// TIA Portal V19 export
FUNCTION "CollectAlarms" : Void   // FC62, LAD
TITLE = Alarm Collector Unit
// Collects alarms from the respective level and categorises the alarms into the different alarm classes. Filling the alarm DB with specific alarm messages which are defined in the comment of the defined alarm. The definition of possible alarms within a equipment is handled here.
// stored: Namespace Unit3.EM1, SetENOAutomatically false
   VAR_INPUT
      resetAlarms : Bool;
      disableAlarms : Bool;
   END_VAR
   VAR_OUTPUT
      commandsToUnit : "LUC_typeStateCommands";   // Feedback to the unit
   END_VAR
   VAR_TEMP   // added for the SCL form of the ladder/FBD networks
      _w1 : Bool;
   END_VAR
BEGIN

REGION Network 1: Reset Alarms
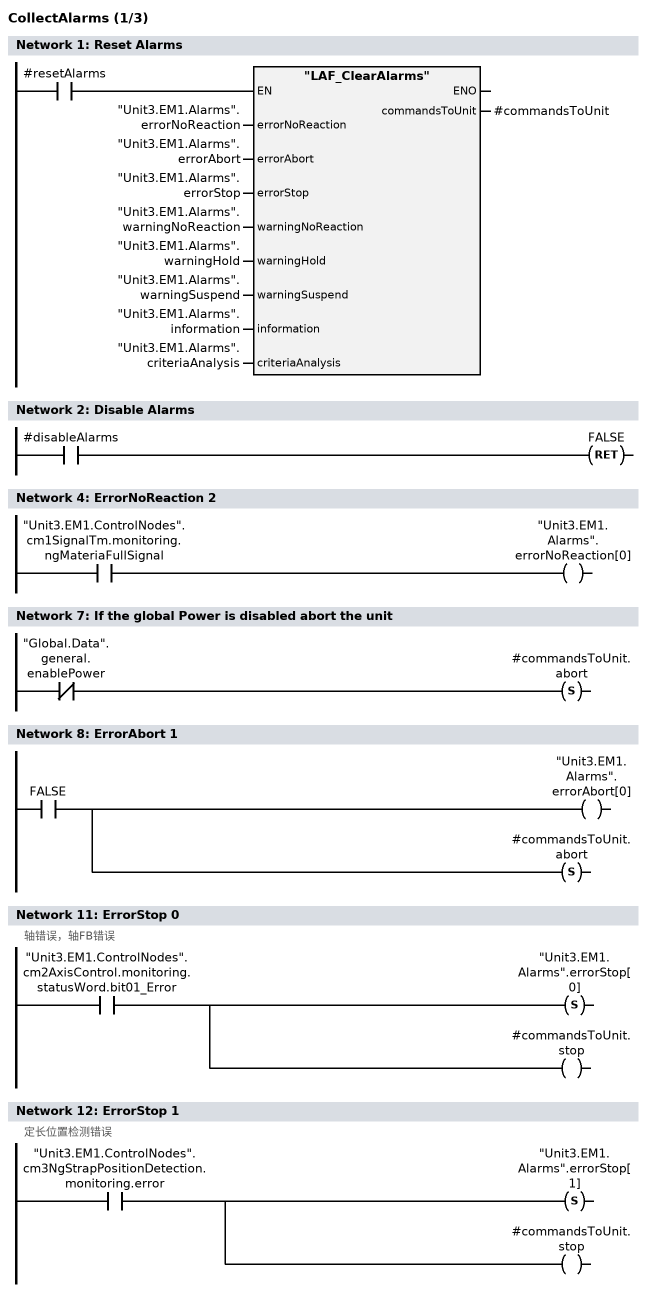
   RUNG wire#powerrail
      Contact( #resetAlarms )
      "LAF_ClearAlarms"(errorNoReaction := "Unit3.EM1.Alarms".errorNoReaction, errorAbort := "Unit3.EM1.Alarms".errorAbort, errorStop := "Unit3.EM1.Alarms".errorStop, warningNoReaction := "Unit3.EM1.Alarms".warningNoReaction, warningHold := "Unit3.EM1.Alarms".warningHold, warningSuspend := "Unit3.EM1.Alarms".warningSuspend, information := "Unit3.EM1.Alarms".information, criteriaAnalysis := "Unit3.EM1.Alarms".criteriaAnalysis, commandsToUnit => #commandsToUnit)
   END_RUNG
   // the same network as SCL:
   IF #resetAlarms THEN
       "LAF_ClearAlarms"(errorNoReaction := "Unit3.EM1.Alarms".errorNoReaction,
                         errorAbort := "Unit3.EM1.Alarms".errorAbort,
                         errorStop := "Unit3.EM1.Alarms".errorStop,
                         warningNoReaction := "Unit3.EM1.Alarms".warningNoReaction,
                         warningHold := "Unit3.EM1.Alarms".warningHold,
                         warningSuspend := "Unit3.EM1.Alarms".warningSuspend,
                         information := "Unit3.EM1.Alarms".information,
                         criteriaAnalysis := "Unit3.EM1.Alarms".criteriaAnalysis,
                         commandsToUnit => #commandsToUnit);
   END_IF;
END_REGION

REGION Network 2: Disable Alarms
   RUNG wire#powerrail
      Contact( #disableAlarms )
      ReturnCoil( FALSE )
   END_RUNG
   // the same network as SCL:
   IF #disableAlarms THEN
       ENO := FALSE;
       RETURN;
   END_IF;
END_REGION

REGION Network 3: *************** Error No Reaction ************************
END_REGION

REGION Network 4: ErrorNoReaction 2
   RUNG wire#powerrail
      Contact( "Unit3.EM1.ControlNodes".cm1SignalTm.monitoring.ngMateriaFullSignal )
      Coil( "Unit3.EM1.Alarms".errorNoReaction[0] )
   END_RUNG
   // the same network as SCL:
   "Unit3.EM1.Alarms".errorNoReaction[0] := "Unit3.EM1.ControlNodes".cm1SignalTm.monitoring.ngMateriaFullSignal;
END_REGION

REGION Network 6: *************** Error and Abort **************************
END_REGION

REGION Network 7: If the global Power is disabled abort the unit
   RUNG wire#powerrail
      I_Contact( "Global.Data".general.enablePower )
      S_Coil( #commandsToUnit.abort )
   END_RUNG
   // the same network as SCL:
   IF NOT "Global.Data".general.enablePower THEN #commandsToUnit.abort := TRUE; END_IF;
END_REGION

REGION Network 8: ErrorAbort 1
   RUNG wire#powerrail
      Contact( FALSE )
      wire#w1
      Coil( "Unit3.EM1.Alarms".errorAbort[0] )
   END_RUNG
   RUNG wire#w1
      S_Coil( #commandsToUnit.abort )
   END_RUNG
   // the same network as SCL:
   "Unit3.EM1.Alarms".errorAbort[0] := FALSE;
   IF FALSE THEN #commandsToUnit.abort := TRUE; END_IF;
END_REGION

REGION Network 10: *************** Error and Stop ***************************
END_REGION

REGION Network 11: ErrorStop 0
   // 轴错误，轴FB错误
   RUNG wire#powerrail
      Contact( "Unit3.EM1.ControlNodes".cm2AxisControl.monitoring.statusWord.bit01_Error )
      wire#w1
      S_Coil( "Unit3.EM1.Alarms".errorStop[0] )
   END_RUNG
   RUNG wire#w1
      Coil( #commandsToUnit.stop )
   END_RUNG
   // the same network as SCL:
   IF "Unit3.EM1.ControlNodes".cm2AxisControl.monitoring.statusWord.bit01_Error THEN
       "Unit3.EM1.Alarms".errorStop[0] := TRUE;
   END_IF;
   #commandsToUnit.stop := "Unit3.EM1.ControlNodes".cm2AxisControl.monitoring.statusWord.bit01_Error;
END_REGION

REGION Network 12: ErrorStop 1
   // 定长位置检测错误
   RUNG wire#powerrail
      Contact( "Unit3.EM1.ControlNodes".cm3NgStrapPositionDetection.monitoring.error )
      wire#w1
      S_Coil( "Unit3.EM1.Alarms".errorStop[1] )
   END_RUNG
   RUNG wire#w1
      Coil( #commandsToUnit.stop )
   END_RUNG
   // the same network as SCL:
   IF "Unit3.EM1.ControlNodes".cm3NgStrapPositionDetection.monitoring.error THEN
       "Unit3.EM1.Alarms".errorStop[1] := TRUE;
   END_IF;
   #commandsToUnit.stop := "Unit3.EM1.ControlNodes".cm3NgStrapPositionDetection.monitoring.error;
END_REGION

REGION Network 13: ErrorStop 2
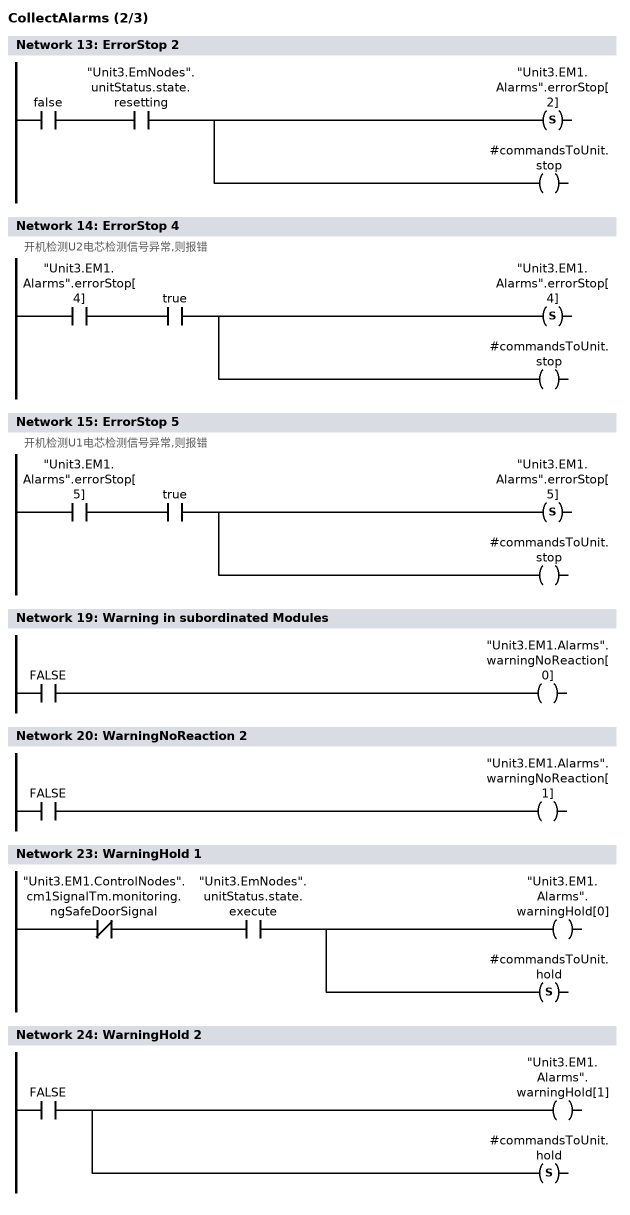
   RUNG wire#powerrail
      Contact( false )
      Contact( "Unit3.EmNodes".unitStatus.state.resetting )
      wire#w1
      S_Coil( "Unit3.EM1.Alarms".errorStop[2] )
   END_RUNG
   RUNG wire#w1
      Coil( #commandsToUnit.stop )
   END_RUNG
   // the same network as SCL:
   #_w1 := false AND "Unit3.EmNodes".unitStatus.state.resetting;
   IF #_w1 THEN "Unit3.EM1.Alarms".errorStop[2] := TRUE; END_IF;
   #commandsToUnit.stop := #_w1;
END_REGION

REGION Network 14: ErrorStop 4
   // 开机检测U2电芯检测信号异常,则报错
   RUNG wire#powerrail
      Contact( "Unit3.EM1.Alarms".errorStop[4] )
      Contact( true )
      wire#w1
      S_Coil( "Unit3.EM1.Alarms".errorStop[4] )
   END_RUNG
   RUNG wire#w1
      Coil( #commandsToUnit.stop )
   END_RUNG
   // the same network as SCL:
   #_w1 := "Unit3.EM1.Alarms".errorStop[4] AND true;
   IF #_w1 THEN "Unit3.EM1.Alarms".errorStop[4] := TRUE; END_IF;
   #commandsToUnit.stop := #_w1;
END_REGION

REGION Network 15: ErrorStop 5
   // 开机检测U1电芯检测信号异常,则报错
   RUNG wire#powerrail
      Contact( "Unit3.EM1.Alarms".errorStop[5] )
      Contact( true )
      wire#w1
      S_Coil( "Unit3.EM1.Alarms".errorStop[5] )
   END_RUNG
   RUNG wire#w1
      Coil( #commandsToUnit.stop )
   END_RUNG
   // the same network as SCL:
   #_w1 := "Unit3.EM1.Alarms".errorStop[5] AND true;
   IF #_w1 THEN "Unit3.EM1.Alarms".errorStop[5] := TRUE; END_IF;
   #commandsToUnit.stop := #_w1;
END_REGION

REGION Network 18: *************** Warning No Reaction **********************
END_REGION

REGION Network 19: Warning in subordinated Modules
   RUNG wire#powerrail
      Contact( FALSE )
      Coil( "Unit3.EM1.Alarms".warningNoReaction[0] )
   END_RUNG
   // the same network as SCL:
   "Unit3.EM1.Alarms".warningNoReaction[0] := FALSE;
END_REGION

REGION Network 20: WarningNoReaction 2
   RUNG wire#powerrail
      Contact( FALSE )
      Coil( "Unit3.EM1.Alarms".warningNoReaction[1] )
   END_RUNG
   // the same network as SCL:
   "Unit3.EM1.Alarms".warningNoReaction[1] := FALSE;
END_REGION

REGION Network 22: *************** Warning Hold **************************
END_REGION

REGION Network 23: WarningHold 1
   RUNG wire#powerrail
      I_Contact( "Unit3.EM1.ControlNodes".cm1SignalTm.monitoring.ngSafeDoorSignal )
      Contact( "Unit3.EmNodes".unitStatus.state.execute )
      wire#w1
      Coil( "Unit3.EM1.Alarms".warningHold[0] )
   END_RUNG
   RUNG wire#w1
      S_Coil( #commandsToUnit.hold )
   END_RUNG
   // the same network as SCL:
   "Unit3.EM1.Alarms".warningHold[0] := NOT "Unit3.EM1.ControlNodes".cm1SignalTm.monitoring.ngSafeDoorSignal AND "Unit3.EmNodes".unitStatus.state.execute;
   IF NOT "Unit3.EM1.ControlNodes".cm1SignalTm.monitoring.ngSafeDoorSignal AND "Unit3.EmNodes".unitStatus.state.execute THEN
       #commandsToUnit.hold := TRUE;
   END_IF;
END_REGION

REGION Network 24: WarningHold 2
   RUNG wire#powerrail
      Contact( FALSE )
      wire#w1
      Coil( "Unit3.EM1.Alarms".warningHold[1] )
   END_RUNG
   RUNG wire#w1
      S_Coil( #commandsToUnit.hold )
   END_RUNG
   // the same network as SCL:
   "Unit3.EM1.Alarms".warningHold[1] := FALSE;
   IF FALSE THEN #commandsToUnit.hold := TRUE; END_IF;
END_REGION

REGION Network 26: *************** Warning Suspend ***********************
END_REGION

REGION Network 27: WarningSuspend 1
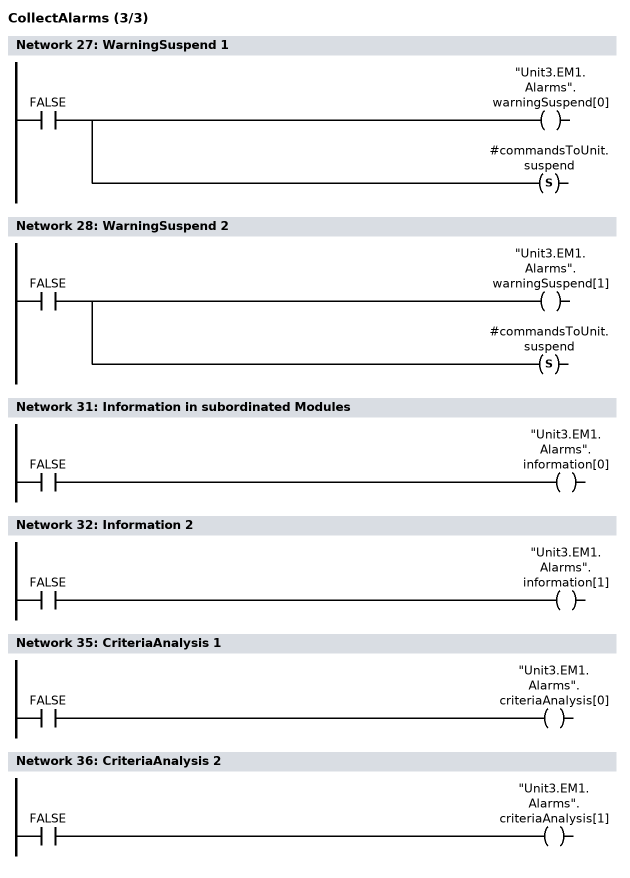
   RUNG wire#powerrail
      Contact( FALSE )
      wire#w1
      Coil( "Unit3.EM1.Alarms".warningSuspend[0] )
   END_RUNG
   RUNG wire#w1
      S_Coil( #commandsToUnit.suspend )
   END_RUNG
   // the same network as SCL:
   "Unit3.EM1.Alarms".warningSuspend[0] := FALSE;
   IF FALSE THEN #commandsToUnit.suspend := TRUE; END_IF;
END_REGION

REGION Network 28: WarningSuspend 2
   RUNG wire#powerrail
      Contact( FALSE )
      wire#w1
      Coil( "Unit3.EM1.Alarms".warningSuspend[1] )
   END_RUNG
   RUNG wire#w1
      S_Coil( #commandsToUnit.suspend )
   END_RUNG
   // the same network as SCL:
   "Unit3.EM1.Alarms".warningSuspend[1] := FALSE;
   IF FALSE THEN #commandsToUnit.suspend := TRUE; END_IF;
END_REGION

REGION Network 30: *************** Information *****************************
END_REGION

REGION Network 31: Information in subordinated Modules
   RUNG wire#powerrail
      Contact( FALSE )
      Coil( "Unit3.EM1.Alarms".information[0] )
   END_RUNG
   // the same network as SCL:
   "Unit3.EM1.Alarms".information[0] := FALSE;
END_REGION

REGION Network 32: Information 2
   RUNG wire#powerrail
      Contact( FALSE )
      Coil( "Unit3.EM1.Alarms".information[1] )
   END_RUNG
   // the same network as SCL:
   "Unit3.EM1.Alarms".information[1] := FALSE;
END_REGION

REGION Network 34: *************** CriteriaAnalysis **************************
END_REGION

REGION Network 35: CriteriaAnalysis 1
   RUNG wire#powerrail
      Contact( FALSE )
      Coil( "Unit3.EM1.Alarms".criteriaAnalysis[0] )
   END_RUNG
   // the same network as SCL:
   "Unit3.EM1.Alarms".criteriaAnalysis[0] := FALSE;
END_REGION

REGION Network 36: CriteriaAnalysis 2
   RUNG wire#powerrail
      Contact( FALSE )
      Coil( "Unit3.EM1.Alarms".criteriaAnalysis[1] )
   END_RUNG
   // the same network as SCL:
   "Unit3.EM1.Alarms".criteriaAnalysis[1] := FALSE;
END_REGION
END_FUNCTION
